// TIA Portal V16 export
// export: Created 2023-08-28T09:37:50.0116378Z, ExportSetting WithDefaults, DisplayName Totally Integrated Automation Portal, DisplayVersion V16 Update 6, DisplayName TIA Portal Version Control Interface, DisplayVersion V16 Update 2, DisplayName TIA Portal Openness, DisplayVersion V16 Update 6, DisplayName STEP 7 Professional, DisplayVersion V16 Update 6, DisplayName STEP 7 Safety, DisplayVersion V16, DisplayName WinCC Advanced, DisplayVersion V16 Update 6
DATA_BLOCK "MB_COMM_LOAD_DB"   // DB34
// stored: AutoNumber true, DBAccessibleFromOPCUA true, InstanceOfName MB_COMM_LOAD, OfSystemLibElement MB_COMM_LOAD, OfSystemLibVersion 2.1
"MB_COMM_LOAD"
   // VAR_INPUT
   //    REQ : Bool;
   //    PORT : PORT;
   //    BAUD : UDInt;
   //    PARITY : UInt;
   //    FLOW_CTRL : UInt;
   //    RTS_ON_DLY : UInt;
   //    RTS_OFF_DLY : UInt;
   //    RESP_TO : UInt;
   // END_VAR
   // VAR_OUTPUT
   //    DONE : Bool;
   //    ERROR : Bool;
   //    STATUS : Word;
   // END_VAR
   // VAR_IN_OUT
   //    MB_DB : MB_BASE;
   // END_VAR
   // VAR
   //    ICHAR_GAP : UInt;
   //    RETRIES : UInt;
   //    WRREC_STATUS : Word;
   //    RDREC_STATUS : Word;
   //    SFC_STATUS : Word;
   //    Port_CFG_SFB : Array[0..25] of Byte;
   //    Send_CFG_SFB : Array[0..16] of Byte;
   //    Rcv_CFG_SFB : Array[0..60] of Byte;
   //    STOP_BITS : USInt := 1;
   // END_VAR
BEGIN
END_DATA_BLOCK
